PROGRAM MAIN
VAR
END_VAR

END_PROGRAM

(* stored: Version 1.1.0.1
   POU MAIN: Id {a58a46ad-6bfb-4454-9977-6eb277d8a129} *)
